TYPE E_TableManager_States : (
	TABLEMANAGER_DISABLED,
	TABLEMANAGER_ENABLING,
	TABLEMANAGER_HOMMING_READY_TO_START,
	TABLEMANAGER_HOMMING,
	TABLEMANAGER_HALT_FEED,

	(* Standard Running States *)
	TABLEMANAGER_IDLE_FEED_OFF,				(* feed off *)
	TABLEMANAGER_CLAMPPING,
	TABLEMANAGER_CLAMPED,
	TABLEMANAGER_UNCLAMP_START,
	TABLEMANAGER_UNCLAMPING,

	(* Auto-feed States *)
	TABLEMANAGER_AUTOFEED_INIT,
	TABLEMANAGER_AUTOFEED_INIT_RESTART,
	TABLEMANAGER_AUTOFEED_IDLE,
	TABLEMANAGER_AUTOFEED_START_DOOR_IN,
	TABLEMANAGER_AUTOFEED_WAIT_FOR_DATA,
	TABLEMANAGER_AUTOFEED_FEEDTHRU_START,
	TABLEMANAGER_AUTOFEED_INSTOP,
	TABLEMANAGER_AUTOFEED_INSTOP_HALT,
	TABLEMANAGER_AUTOFEED_INSTOP_BACK_TO_STOP,
	TABLEMANAGER_AUTOFEED_OUTSTOP,
	TABLEMANAGER_AUTOFEED_OUTSTOP_SLOW,
//	TABLEMANAGER_AUTOFEED_OUTSTOP_AT_STOP,
//	TABLEMANAGER_AUTOFEED_OUTSTOP_NEW_TARGET,
	TABLEMANAGER_AUTOFEED_FEED_OUT,
	TABLEMANAGER_AUTOFEED_FEED_OUT_PAUSED,
	TABLEMANAGER_AUTOFEED_FEED_OUT_DONE,
	TABLEMANAGER_AUTOFEED_RE_FEED_BACK_TO_STOP,
	(* Refeed Sequence *)
	TABLEMANAGER_REFEED_START,
	TABLEMANAGER_REFEED_WAIT_FOR_CONTINUE,
	TABLEMANAGER_REFEED_UNCLAMP,
	TABLEMANAGER_REFEED_TO_INFEED,
//	TABLEMANAGER_REFEED_TO_OUTFEED_MOVE_STOP,
	TABLEMANAGER_REFEED_TO_OUTFEED,
	(* Reset Sequence *)
	TABLEMANAGER_RESET_INIT,
	TABLEMANAGER_RESETTING,
	TABLEMANAGER_RESET_DONE,

	(* Error States *)
	TABLEMANAGER_ERROR
);
END_TYPE

(* stored: Version 1.1.0.1, ProductVersion 3.1.4024.13
   DUT E_TableManager_States: Id {a9a00e66-6cdd-472c-9fc7-66a9a3b8be26} *)
